(*
version 1.0	4 Feb 2007
programmer 	hugo
tested by		tobias

this function converts velocities from Meters / Second to Kilometers / hour.

*)
FUNCTION MS_TO_KMH : REAL
VAR_INPUT
	ms : REAL;
END_VAR

MS_TO_KMH := ms * 3.6;

END_FUNCTION

(* stored: Version 1.1.0.1
   POU MS_TO_KMH: Id {51fdfa69-2063-4fa3-b54e-caf20b6a2a72}, SpecialFunc None *)
